PROGRAM P_GroupsWcStates
VAR_INPUT
	bReset															: BOOL;
	arrWcStateSyncUnitGroup	 				AT %I* 					: ARRAY [1..iNumberOfSyncUnitGroups] OF BOOL; (*Link to SyncUnit WcStates*)
END_VAR

VAR_OUTPUT
	bOK																: BOOL;
	bError															: BOOL;
	udiErrorID														: UDINT;
	sErrorDescription												: WSTRING;
END_VAR                                                     		
                                                            		
VAR                                                         	
	rtReset															: R_TRIG;
	bFirstCycle														: BOOL;
END_VAR                                                     	
                                                            	
VAR CONSTANT                                                	
	iNumberOfSyncUnitGroups											: INT:= 9;					// Deklaracja liczby grup SyncUnit
END_VAR

IF iNumberOfSyncUnitGroups = 0 OR NOT bFirstCycle THEN
	bFirstCycle															:= TRUE;
	RETURN;
END_IF

rtReset(CLK:= bReset);

FOR i:= 1 TO iNumberOfSyncUnitGroups DO
	IF arrWcStateSyncUnitGroup[i] THEN
		bError														:= TRUE;
		EXIT;                                               		
	END_IF                                                  		
END_FOR                                                     		
                                                            		
bOK																	:= NOT bError;	
                                                            		
                                                            		
IF arrWcStateSyncUnitGroup[1] THEN                          		
	udiErrorID														:= 84;
	sErrorDescription												:= "Błąd sterownika | Błąd komunikacji modułów komunikacyjnych";
END_IF   

IF arrWcStateSyncUnitGroup[2] THEN                          		
	udiErrorID														:= 85;
	sErrorDescription												:= "Błąd sterownika | Błąd komunikacji modułów I/O";
END_IF                                                 			
                                                        			
IF arrWcStateSyncUnitGroup[3] THEN                      			
	udiErrorID														:= 86;
	sErrorDescription												:= "Błąd sterownika | Błąd komunikacji grupy falowników";
END_IF 
                                                 		
IF arrWcStateSyncUnitGroup[4] THEN                      			
	udiErrorID														:= 87;
	sErrorDescription												:= "Błąd sterownika | Błąd komunikacji grupy modułów safety";
END_IF  
                                                      		
IF arrWcStateSyncUnitGroup[5] THEN                      			
	udiErrorID														:= 88;
	sErrorDescription												:= "Błąd sterownika | Błąd komunikacji grupy modułów pneumatycznych";
END_IF   

IF arrWcStateSyncUnitGroup[6] THEN                      			
	udiErrorID														:= 89;
	sErrorDescription												:= "Błąd sterownika | Błąd komunikacji grupy safety NC";
END_IF 

IF arrWcStateSyncUnitGroup[7] THEN                      			
	udiErrorID														:= 90;
	sErrorDescription												:= "Błąd sterownika | Błąd komunikacji grupy analogowych";
END_IF   
                                                  		
IF rtReset.Q THEN                                       		
	bError															:= FALSE;
	udiErrorID														:= 0;
	sErrorDescription												:= "";
END_IF

END_PROGRAM

(* stored: Version 1.1.0.1, ProductVersion 3.1.4026.13, FileIdentifier 0c62d254aa0ca576ddc26306493d11fe815c5cdf, FileSignature 0801296022bcc3d2fb710f1df0865a1379d8183d1f667e17b103aa6ef9fc18a75ce7bf709b898e4917bdffd52a1141a004d0d6cb0dca931b46fa2ef53f68a7f569e0bc092512e3ffbb132ec6a15f393a4f8b8d55e3155d48581f1413a53fdebba4d5a340a5f0c56e8a6e7a2fcbba175bcc8843cf17019b5a759e2d1913e1b2e0a45317449e8546fddeec10b522555619cba77eb8c9916f5b2eec88e655014617bafece55ef8bfde8cad175c805f18c075adf51746700582299e3413067d61aec49bccff376a2e622680bb1596fc38ccf4dc9a58f7d4b5987dcf4ad6f3a53c842671d024f8caefd90e6e494ad3ab0d82aaee84ac23be9a7d2a817e05a5b9b1216
   POU P_GroupsWcStates: Id {802eace0-b31e-468f-bd0f-4ef4d4a3ff64}, SpecialFunc None *)
